// TIA Portal project "Traffic_Light" (V18)

(* hardware
DEVICE "S7-1200 station_1"  S7-1200 Station
   slot 0: "Rack_0"  S7-1200 Rack  Rack  V1.0
   slot 1: "PLC_1"  CPU 1214C DC/DC/DC  6ES7 214-1AG40-0XB0  V4.6
*)

// ===== PLC "PLC_1"  CPU 1214C DC/DC/DC =====

VAR_GLOBAL   // PLC tag table "Default tag table"
   "T0" AT %MD6 : Time;
   "T1" AT %MD10 : Time;
END_VAR

VAR_GLOBAL   // PLC tag table "Output"
   "Green_Led" AT %Q0.0 : Bool;
   "Red_Led" AT %Q0.1 : Bool;
   "Yellow_Led" AT %Q0.2 : Bool;
END_VAR

VAR_GLOBAL   // PLC tag table "Memory"
   "Run_Mode" AT %M0.0 : Bool;
   "Repeat_Cycle" AT %M0.1 : Bool;
END_VAR

VAR_GLOBAL   // PLC tag table "Inputs"
   "Start" AT %I0.0 : Bool;
   "Reset" AT %I0.1 : Bool;
   "Traffic_Sensor" AT %I0.2 : Bool;
END_VAR

// folder: System blocks/Program resources

DATA_BLOCK "IEC_Timer_0_DB"   // DB1
{ S7_Optimized_Access := 'TRUE' }
AUTHOR : Simatic
FAMILY : IEC
NAME : IEC_TMR
VERSION : 1.0
// stored: InstanceOfName IEC_TIMER
"IEC_TIMER"
BEGIN
END_DATA_BLOCK

DATA_BLOCK "IEC_Timer_0_DB_1"   // DB2
{ S7_Optimized_Access := 'TRUE' }
AUTHOR : Simatic
FAMILY : IEC
NAME : IEC_TMR
VERSION : 1.0
// stored: InstanceOfName IEC_TIMER
"IEC_TIMER"
BEGIN
END_DATA_BLOCK

DATA_BLOCK "IEC_Timer_0_DB_2"   // DB3
{ S7_Optimized_Access := 'TRUE' }
AUTHOR : Simatic
FAMILY : IEC
NAME : IEC_TMR
VERSION : 1.0
// stored: InstanceOfName IEC_TIMER
"IEC_TIMER"
BEGIN
END_DATA_BLOCK

// folder: (top level)

ORGANIZATION_BLOCK "Main"   // OB1, LAD, ProgramCycle
TITLE = "Main Program Sweep (Cycle)"
{ S7_Optimized_Access := 'TRUE' }
VERSION : 0.1
   VAR_INPUT
      Initial_Call : Bool;   // Initial call of this OB
      Remanence : Bool;   // =True, if remanent data are available
   END_VAR
BEGIN

REGION Network 1
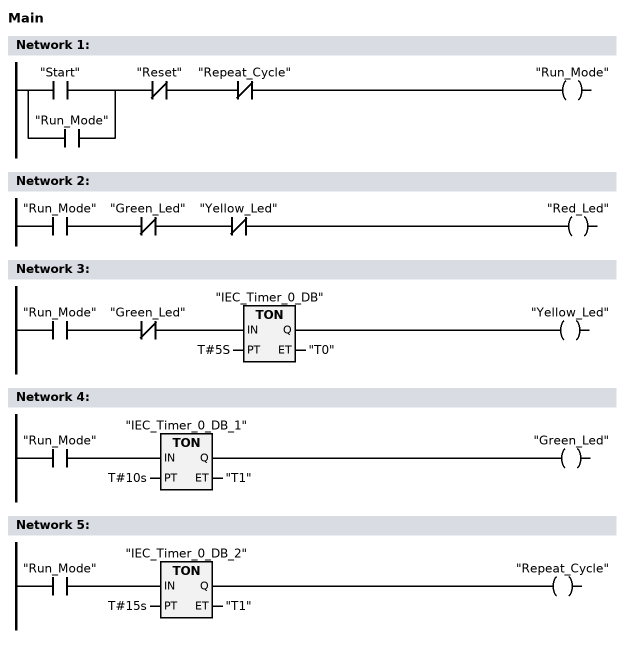
   RUNG wire#powerrail
      Contact( "Start" )
      wire#w1
      I_Contact( "Reset" )
      I_Contact( "Repeat_Cycle" )
      Coil( "Run_Mode" )
   END_RUNG
   RUNG wire#powerrail
      Contact( "Run_Mode" )
   END_RUNG wire#w1
   // the same network as SCL:
   "Run_Mode" := ("Start" OR "Run_Mode") AND NOT "Reset" AND NOT "Repeat_Cycle";
END_REGION

REGION Network 2
   RUNG wire#powerrail
      Contact( "Run_Mode" )
      I_Contact( "Green_Led" )
      I_Contact( "Yellow_Led" )
      Coil( "Red_Led" )
   END_RUNG
   // the same network as SCL:
   "Red_Led" := "Run_Mode" AND NOT "Green_Led" AND NOT "Yellow_Led";
END_REGION

REGION Network 3
   "IEC_Timer_0_DB".TON(IN := "Run_Mode" AND NOT "Green_Led", PT := T#5S, ET => "T0");
   "Yellow_Led" := "IEC_Timer_0_DB".Q;
END_REGION

REGION Network 4
   "IEC_Timer_0_DB_1".TON(IN := "Run_Mode", PT := T#10s, ET => "T1");
   "Green_Led" := "IEC_Timer_0_DB_1".Q;
END_REGION

REGION Network 5
   "IEC_Timer_0_DB_2".TON(IN := "Run_Mode", PT := T#15s, ET => "T1");
   "Repeat_Cycle" := "IEC_Timer_0_DB_2".Q;
END_REGION
END_ORGANIZATION_BLOCK